PROGRAM MAIN
VAR
	Manual_Automatic:BOOL;
	Visible:BOOL;
END_VAR

Stop();
Emergency_Stop();
Automatic_Or_Manual();
Visible:=not gvl.ixA;

END_PROGRAM

(* stored: Version 1.1.0.1, ProductVersion 3.1.4024.12
   POU MAIN: Id {99369a3d-4dc6-470f-a43b-a616750e939a}, SpecialFunc None *)
